FUNCTION_BLOCK WoodBunkEx
VAR_IN_OUT //controls
	execute : BOOL;
	stop : BOOL;
	
	manualStep : BOOL;
	manualSuction : BOOL;
END_VAR
VAR_IN_OUT //references to required hardware
	robotLeft, robotRight : RobotA21;
	toolStorageLeft, toolStorageRight : A21ToolStorage;
	
	stagingTableLeft, stagingTableRight : StagingTable;
	magazineLeft, magazineRight : SkidMagazine;
	
	strapper : StrapMachine;
	
	horizontalDriveLeft, horizontalDriveRight : AirPiston;
	verticalDriveLeft, verticalDriveRight : ClearLinkMC;
	pistonBottom : SimplePiston;
	
	suctionTop : ARRAY[*] OF SuctionPad; (*1..3*)
	suctionLeft : ARRAY[*] OF SuctionPad; (*1..4*)
	suctionRight : ARRAY[*] OF SuctionPad; (*1..4*)
	suctionBottom : ARRAY[*] OF SuctionPad; (*1..2*)
END_VAR
VAR_OUTPUT
	//ready : BOOL;
	done : BOOL;
	
	generalError : BOOL;
	errorLeft, errorRight : BOOL;
END_VAR
VAR //for testing, to be removed when deployoed
	latchLeft, latchRight : BOOL; //prevents SMC sliders from overshooting the inner limit sensor
	
	suctionEnableTop : BOOL;
	suctionEnableLeft : BOOL;
	suctionEnableRight : BOOL;
	suctionEnableBottom : BOOL;
END_VAR
VAR	
	topSuctionDelay : TON;
	
	step : (IDLE, STAGING, LOAD_WB, PUSH, STRAP, RELEASE, COMPLETE := 1050);
	iPair : INT;
	//these 2 ints should replace the 4 ints after
	masterStep : INT;
	subStepLeft, subStepRight : INT;
	
	loadSet : INT;
	loadStepLeft, loadStepRight : INT;
	
	stageSet : INT;	
	stageStepLeft, stageStepRight : INT;
	iSlotLeft, iSlotRight : INT;
END_VAR
VAR //local types
	demoHeight : REAL := 600; //mm
	materialsArr : ARRAY[0..GVL.maxPairs] OF PositionMaterials := [
		(
			position := 0,
			top := 'WDS20', left := 'WDS20', right := 'WDS20', bottom := 'WDB20'
		),
		(
			position := 69,
			top := 'WDS20', left := 'WDS20', right := 'WDS20', bottom := 'WDB20'
		)];
	
	templateSlotsLeft, templateSlotsRight : ARRAY[1..10] OF STRING;
	templateOccupancyLeft, templateOccupancyRight : ARRAY[1..10] OF BOOL;
	stagingTemplateLeft, stagingTemplateRight AT %M* : StagingTable;	
	stagingArrayLeft, stagingArrayRight : ARRAY[0..(GVL.maxPairs+1)*2] OF STRING;
	
	insertionLeft, insertionRight : Insertion;
	loadedMaterials : ARRAY[Surface.TOP..Surface.BOTTOM] OF STRING;
END_VAR
VAR CONSTANT
	sectionID : SectionEnum := SectionEnum.WOOD_BUNK;
END_VAR
VAR
	a,b,c,d : BOOL;
	suctionTimerLeft, suctionTimerRight : TON;
END_VAR

callLocalModules(); //initialize local modules

IF stop THEN
	stopSequence(); //stop everything
	RETURN;
END_IF
(*
IF NOT insertionLeft.screw.HomeSet OR NOT insertionRight.screw.HomeSet THEN
	homingSequence(); //homing all motion devices and robots
	RETURN;
END_IF
*)
a S= suctionTop[1].occupied AND suctionTop[2].occupied AND suctionTop[3].occupied;
b S= suctionLeft[1].occupied AND suctionLeft[2].occupied AND suctionLeft[3].occupied AND suctionLeft[4].occupied;
c S= suctionRight[1].occupied AND suctionRight[2].occupied AND suctionRight[3].occupied AND suctionRight[4].occupied;
d S= suctionBottom[1].occupied AND suctionBottom[2].occupied;

CASE step OF
	IDLE:
		IF execute THEN
			execute := FALSE;
			suctionEnableTop := suctionEnableLeft := suctionEnableRight := suctionEnableBottom := FALSE;
			step := STAGING;
		END_IF
		
		SetSuctions(suctionTop, suctionEnableTop);
		SetSuctions(suctionLeft, suctionEnableLeft);
		SetSuctions(suctionRight, suctionEnableRight);
		SetSuctions(suctionBottom, suctionEnableBottom);
		
	STAGING:
		IF NOT done THEN
			done := stage(error => generalError);
		END_IF
		
		IF
			(manualStep AND_THEN execute) OR
			(NOT manualStep AND_THEN done)
		THEN
			execute := FALSE;
			done := FALSE;
			step := LOAD_WB;
		END_IF
	
	LOAD_WB:
		IF NOT done THEN
			done := load(pairIndex := iPair, error => generalError);
		END_IF
		
		IF manualSuction THEN
			SetSuctions(suctionTop, suctionEnableTop);
			SetSuctions(suctionLeft, suctionEnableLeft);
			SetSuctions(suctionRight, suctionEnableRight);
			SetSuctions(suctionBottom, suctionEnableBottom);
		END_IF
		
		IF
			(manualStep AND_THEN execute) OR
			(NOT manualStep AND_THEN done)
		THEN
			done := FALSE;
			suctionEnableTop := suctionEnableLeft := suctionEnableRight := suctionEnableBottom := FALSE;
			execute := FALSE;
			
			step := PUSH;
		END_IF
		
	PUSH:
		IF
			(manualStep AND_THEN execute) OR
			(latchLeft AND latchRight AND pistonBottom.extended)
		THEN
			latchLeft := latchRight := FALSE;
			execute := FALSE;
			step := STRAP;
			RETURN;
		END_IF
		
		IF NOT validateSuctionQuality(checkTop:= TRUE, checkLeft:= TRUE, checkRight:= FALSE, checkBottom:= FALSE) THEN
			generalError := TRUE;
			RETURN;
		END_IF
		(*
		IF 
			insertionLeft.sliderPos <> demoHeight/2 //OR 
			//insertionRight.sliderPos <> demoHeight/2 //OR 
			//NOT insertionBottom.contact
		THEN
			insertionLeft.slideAbsolute(demoHeight/2);
			//insertionRight.slideAbsolute(demoHeight/2);
			RETURN;
		END_IF
		*)
		
		IF insertionLeft.screw.AtInnerLimit THEN
			latchLeft := TRUE;
		ELSIF NOT latchLeft THEN
			insertionLeft.press();
		END_IF
		
		IF insertionRight.screw.AtInnerLimit THEN
			latchRight := TRUE;
		ELSIF NOT latchRight THEN
			insertionRight.press();
		END_IF
		pistonBottom.extend();
		
	STRAP:
		topSuctionDelay(IN:= , PT:= T#1S, Q=> , ET=> );
		
		strapper.bEnable := TRUE;
		IF strapper.done THEN
			topSuctionDelay.IN := FALSE;
			step := RELEASE;
			RETURN;
		END_IF
		
		IF topSuctionDelay.Q THEN
			SetSuctions(suctionTop, FALSE);
			SetSuctions(suctionLeft, FALSE);
			SetSuctions(suctionRight, FALSE);
			SetSuctions(suctionBottom, FALSE);
		ELSIF strapper.atBundleLevel THEN
			topSuctionDelay.IN := TRUE;
		END_IF
		
		IF strapper.ready THEN
			strapper.strap();
		END_IF
		
		IF execute THEN
			topSuctionDelay.IN := FALSE;
			execute := FALSE;
			step := RELEASE;
		END_IF
		
	RELEASE: //release command		
		//insertionLeft.slideAbsolute(0);
		//insertionRight.slideAbsolute(0);
		
		insertionLeft.release();
		insertionRight.release();
		pistonBottom.retract();
		
		IF 
			(insertionLeft.screw.AtHome AND insertionRight.screw.AtHome AND pistonBottom.retracted) OR
			execute
		THEN
			execute := FALSE;
			step := COMPLETE;
		END_IF
	
	COMPLETE:
		//reset everything
		iPair := (iPair + 1) MOD GVL.maxPairs;
		step := IDLE;
		a := b := c := d := FALSE;
END_CASE

ACTION callLocalModules:
{warning disable C0371}
stagingTemplateLeft(slots := templateSlotsLeft, occupied := templateOccupancyLeft);
stagingTemplateRight(slots := templateSlotsRight, occupied := templateOccupancyRight);

insertionLeft(
	enable:= TRUE, 
	slider:= verticalDriveLeft, 
	screw:= horizontalDriveLeft, 
	contact=> , 
	softContact=> , 
	busy=> , 
	error=> , 
	home=> , 
	homingComplete=> , 
	sliderPos=> );
	
insertionRight(
	enable:= TRUE, 
	slider:= verticalDriveRight, 
	screw:= horizontalDriveRight,  
	contact=> , 
	softContact=> , 
	busy=> , 
	error=> , 
	home=> , 
	homingComplete=> , 
	sliderPos=> );
END_ACTION

METHOD createStagingArrayLeft : BOOL
VAR
	remainingMaterial : STRING;
	splitMaterial : STRING;
	
	i : INT;
END_VAR
FOR i:=0 TO GVL.maxPairs BY 1 DO
	remainingMaterial := materialsArr[i].top;
	WHILE FIND(remainingMaterial, '_') > 0 DO
		splitCombinedMaterials(remainingMaterial, splitMaterial);
		IF splitMaterial <> '' THEN
			AddToStringArray(arr := stagingArrayLeft, newString := splitMaterial, numElements => , nextIndex => );
		END_IF
	END_WHILE
	
	IF remainingMaterial <> '' THEN
		AddToStringArray(arr := stagingArrayLeft, newString := remainingMaterial, numElements => , nextIndex => );
	END_IF
	
	
	remainingMaterial := materialsArr[i].left;
	WHILE FIND(remainingMaterial, '_') > 0 DO
		splitCombinedMaterials(remainingMaterial, splitMaterial);
		IF splitMaterial <> '' THEN
			AddToStringArray(arr := stagingArrayLeft, newString := splitMaterial, numElements => , nextIndex => );
		END_IF
	END_WHILE
	
	IF remainingMaterial <> '' THEN
		AddToStringArray(arr := stagingArrayLeft, newString := remainingMaterial, numElements => , nextIndex => );
	END_IF
END_FOR
END_METHOD

METHOD createStagingArrayRight : BOOL
VAR
	remainingMaterial : STRING;
	splitMaterial : STRING;
	
	i : INT;
END_VAR
FOR i:=0 TO GVL.maxPairs*2 BY 1 DO
	remainingMaterial := materialsArr[i].bottom;
	WHILE FIND(remainingMaterial, '_') > 0 DO
		splitCombinedMaterials(remainingMaterial, splitMaterial);
		IF splitMaterial <> '' THEN
			AddToStringArray(arr := stagingArrayRight, newString := splitMaterial, numElements => , nextIndex => );
		END_IF
	END_WHILE
	
	IF remainingMaterial <> '' THEN
		AddToStringArray(arr := stagingArrayRight, newString := remainingMaterial, numElements => , nextIndex => );
	END_IF
	
	
	
	remainingMaterial := materialsArr[i].right;
	WHILE FIND(remainingMaterial, '_') > 0 DO
		splitCombinedMaterials(remainingMaterial, splitMaterial);
		IF splitMaterial <> '' THEN
			AddToStringArray(arr := stagingArrayRight, newString := splitMaterial, numElements => , nextIndex => );
		END_IF
	END_WHILE
	
	IF remainingMaterial <> '' THEN
		AddToStringArray(arr := stagingArrayRight, newString := remainingMaterial, numElements => , nextIndex => );
	END_IF
END_FOR
END_METHOD

METHOD PROTECTED generateStagingTemplate : BOOL
VAR
	remainingMaterial : STRING;
	splitMaterial : STRING;
	
	i : INT;
END_VAR
VAR_STAT
	temp : INT;
END_VAR
createStagingArrayLeft();
createStagingArrayRight();

//AddToStringArray(arr := stagingArrayLeft, newString := 'WDB20', numElements =>, nextIndex => );

(*
iterate through all pairs and autofill the template
replace succesfully autofilled materials with empty string

when staging needs to be performed a 2nd time, autofilling empty strings is always unsuccessful
*)
FOR i:=0 TO GVL.maxPairs*2 BY 1 DO
	IF stagingTemplateLeft.autofill(materialID := stagingArrayLeft[i]) THEN
		stagingArrayLeft[i] := '';
	END_IF
	
	IF stagingTemplateRight.autofill(materialID := stagingArrayRight[i]) THEN
		stagingArrayRight[i] := '';
	END_IF
END_FOR

(*
stagingTemplateLeft.autofill(demoPairWB.top);
stagingTemplateLeft.autofill(demoPairWB.left);

stagingTemplateRight.autofill(demoPairWB.right);
stagingTemplateRight.autofill(demoPairWB.bottom);
*)

generateStagingTemplate := TRUE;
END_METHOD

ACTION homingSequence:
insertionLeft.homingSequence();
insertionRight.homingSequence();
pistonBottom.retract();
END_ACTION

METHOD PROTECTED load : BOOL
VAR_INPUT
	pairIndex : INT;
END_VAR
VAR_OUTPUT
	error : BOOL;
END_VAR
VAR
	pair : REFERENCE TO PositionMaterials REF= materialsArr[pairIndex];
END_VAR
{warning disable C0371}

IF robotLeft.error OR robotRight.error THEN
	error := TRUE;
	RETURN;
	
ELSIF NOT robotLeft.reserve(sectionID) OR NOT robotRight.reserve(sectionID) THEN //loading requires both robots be reserved together
	RETURN;
	
ELSIF //robots have wrong tool
	(robotLeft.tool <> sectionID AND_THEN NOT robotLeft.changeEOAT(targetTool := sectionID)) OR
	(robotRight.tool <> sectionID AND_THEN NOT robotRight.changeEOAT(targetTool := sectionID))
THEN
	RETURN;
END_IF

CASE loadSet OF
	0: //top and bottom
		IF 
			loadingSequence(
				robot:= robotLeft, 
				table:= stagingTableLeft, 
				loadStep:= loadStepLeft, 
				slot:= iSlotLeft,
				suctions:= suctionTop,
				suctionTimer:= suctionTimerLeft,
				surfaceID:= Surface.TOP, 
				material:= pair.top, 
				fail=> errorLeft)
			
			AND
			loadingSequence(
				robot:= robotRight,
				table:= stagingTableRight, 
				loadStep:= loadStepRight, 
				slot:= iSlotRight,
				suctions:= suctionBottom,
				suctionTimer:= suctionTimerRight,
				surfaceID:= Surface.BOTTOM, 
				material:= pair.bottom, 
				fail=> errorRight)
			
		THEN
			suctionTimerLeft.IN := suctionTimerRight.IN := FALSE;
			loadStepLeft := loadStepRight := 0;
			loadSet := 10;
		END_IF
		
	10: //sides
		IF
			loadingSequence(
				robot:= robotLeft, 
				table:= stagingTableLeft, 
				loadStep:= loadStepLeft, 
				slot:= iSlotLeft,
				suctions:= suctionLeft,
				suctionTimer:= suctionTimerLeft,
				surfaceID:= Surface.LEFT, 
				material:= pair.left, 
				fail=> errorLeft)
			
			AND
			loadingSequence(
				robot:= robotRight, 
				table:= stagingTableRight, 
				loadStep:= loadStepRight, 
				slot:= iSlotRight,
				suctions:= suctionRight,
				suctionTimer:= suctionTimerRight,
				surfaceID:= Surface.RIGHT, 
				material:= pair.right, 
				fail=> errorRight)
		THEN
			suctionTimerLeft.IN := suctionTimerRight.IN := FALSE;
			loadStepLeft := loadStepRight := 0;
			loadSet := COMPLETE;
		END_IF
		
	COMPLETE:
		suctionTimerLeft.IN := suctionTimerRight.IN := FALSE;
		
		loadSet := 0;
		loadStepLeft := loadStepRight := 0;
		
		robotLeft.release(sectionID);
		robotRight.release(sectionID);
		
		load := TRUE;
END_CASE
END_METHOD

METHOD loadingSequence : BOOL
VAR_IN_OUT
	robot : RobotA21;
	table : StagingTable;
	suctions : ARRAY[*] OF SuctionPad;
	loadStep : INT;
	slot : INT;
	
	suctionTimer : TON;
END_VAR
VAR_INPUT
	surfaceID : Surface;
	material : STRING;
END_VAR
VAR_OUTPUT
	fail : BOOL;
END_VAR
VAR
	recoveryMagazine : REFERENCE TO SkidMagazine;
	recoveryStageStep : REFERENCE TO INT;
	suctionDelay : TIME := T#2S;
END_VAR
{warning disable C0371}
IF material = '' THEN
	robot.clearCommand();
	loadingSequence := TRUE;
	RETURN;
END_IF

CASE loadStep OF
	0: //wait for robot
		robot.clearCommand();
		IF robot.Ready THEN
			loadStep := 10;
			slot := 0;
		END_IF
		
	10: //grab from table
		IF slot < 1 AND_THEN NOT table.findSlot(materialID := material, atPosition => slot) THEN 
			fail := TRUE;
			RETURN;
		END_IF
		
		IF NOT table.isOccupied(i := slot) AND table.getSlot(i := slot) <> '' THEN //move from table to robot gripper
			robot.HoldMaterial := table.getSlot(i := slot);
			table.remove(i := slot, materialID => );
		END_IF
		
		IF robot.Done THEN
			loadStep := COMPLETE;
			RETURN;
		ELSIF robot.materialAtHoldingPosition >= 1 AND robot.materialAtHoldingPosition <= 8 THEN
			loadStep := 20;
			RETURN;
		END_IF
		
		CASE surfaceID OF
			Surface.TOP: 					robot.setGroup(group := 1, value := A21.LOAD_BUNK_TOP); 
			Surface.LEFT, Surface.RIGHT: 	robot.setGroup(group := 1, value := A21.LOAD_BUNK_SIDE);
			Surface.BOTTOM: 				robot.setGroup(group := 1, value := A21.LOAD_BUNK_BOTTOM);
		END_CASE
		robot.setGroup(group := 2, value := slot); 
			
	20: //place to insertion
		IF robot.materialAtHoldingPosition > 0 AND robot.HoldMaterial <> '' THEN //move from gripper to insertion
			IF loadedMaterials[surfaceID] = '' THEN //transfer to insertion as is
				loadedMaterials[surfaceID] := robot.HoldMaterial;
			ELSE //join with existing material using underscore _
				loadedMaterials[surfaceID] := JoinStrings(loadedMaterials[surfaceID], robot.HoldMaterial, '_');
			END_IF
			robot.HoldMaterial := '';
		END_IF
		
		CASE surfaceID OF
			Surface.TOP, Surface.BOTTOM:
				SetSuctions(suctions, TRUE (*robot.materialAtHoldingPosition = 1 OR robot.materialAtHoldingPosition = 4*));
				
			Surface.LEFT, Surface.RIGHT:
				SetSuctions(suctions, TRUE (*robot.materialAtHoldingPosition = 2 OR robot.materialAtHoldingPosition = 3*));
				(*
				FOR i:=LOWER_BOUND(suctions, 1) TO UPPER_BOUND(suctions, 1) BY 1 DO
					
					IF i < UPPER_BOUND(suctions, 1)/2 THEN
						suctions[i].enable := robot.materialAtHoldingPosition = 2; //enable upper half suctions
					ELSE
						suctions[i].enable := robot.materialAtHoldingPosition = 3; //enable lower half suctions
					END_IF

				END_FOR
				*)
		END_CASE
		
		suctionTimer(IN:= , PT:= suctionDelay, Q=> , ET=> );
		suctionTimer.IN := TRUE;
		IF NOT suctionTimer.Q THEN
			RETURN;
		END_IF
		
		IF robot.Done THEN
			suctionTimer.IN := FALSE;
			loadStep := COMPLETE;
		END_IF
		
		robot.setGroup(group := 9, value := robot.materialAtHoldingPosition);
	
	COMPLETE:
		robot.clearCommand();
		
		//check insertion quality
		suctionTimer(IN:= , PT:= suctionDelay, Q=> , ET=> );
		suctionTimer.IN := TRUE;
		IF NOT suctionTimer.Q THEN
			RETURN;
		END_IF
		
		IF InsertionQuality(suctions := suctions, insertionMaterial := loadedMaterials[surfaceID], recipeMaterial := material) THEN
			loadingSequence := TRUE;
		ELSE //recovery - remove, restage, and reload
			suctionTimer.IN := FALSE;
			loadStep := 100;
			
		END_IF
		
	100:
		robot.clearCommand();
		IF robot.Ready THEN
			loadStep := 110;
		END_IF
		
	110: //recovery - remove from insertion
		IF robot.Done THEN
			loadStep := 120;
			RETURN;
		END_IF
		
		CASE surfaceID OF
			Surface.TOP:					robot.setGroup(group := 1, value := A21.REMOVE_BUNK_TOP);
			Surface.LEFT, Surface.RIGHT:	robot.setGroup(group := 1, value := A21.REMOVE_BUNK_SIDE);
			Surface.BOTTOM:					robot.setGroup(group := 1, value := A21.REMOVE_BUNK_BOTTOM);
		END_CASE
		
	120:
		robot.clearCommand();
		IF robot.Ready THEN
			loadStep := 130;
		END_IF
		
	130: //recovery - restage
		CASE surfaceID OF
			Surface.TOP, Surface.LEFT:
				recoveryMagazine REF= magazineLeft;			
				recoveryStageStep REF= stageStepLeft;
				
			Surface.RIGHT, Surface.BOTTOM:
				recoveryMagazine REF= magazineRight;			
				recoveryStageStep REF= stageStepRight;
				
		END_CASE
		
		IF
			stageSingle(
				robot:= robot, 
				table:= table, 
				magazine:= recoveryMagazine, 
				stageStep:= recoveryStageStep, 
				slot:= slot, 
				material:= material, 
				fail=> fail)
		THEN
			SetSuctions(suctionPads := suctions, state := FALSE);
			loadStep := 0; //retry
		END_IF
	
END_CASE
END_METHOD

METHOD splitCombinedMaterials : BOOL
VAR_IN_OUT
	materialID : STRING;
	splitMaterial : STRING;
END_VAR
VAR
	i : INT;
END_VAR
FindAndSplitChar(
	sSeparatorChar:= '_', 
	pSrcString:= ADR(materialID), 
	
	pLeftString:= ADR(splitMaterial), 
	nLeftSize:= SIZEOF(splitMaterial), 
	
	pRightString:= ADR(materialID), 
	nRightSize:= SIZEOF(materialID), 
	
	bSearchFromRight:= FALSE);
END_METHOD

METHOD stage : BOOL
VAR_OUTPUT
	error : BOOL;
END_VAR
VAR_STAT
	temp : ARRAY[1..4] OF BOOL;
	boundsErr : ARRAY[1..4] OF BOOL;
END_VAR
{warning disable C0371}
temp[1] := stagingTableLeft.isOccupied(i := 1, errorBounds => boundsErr[1]);
temp[2] := stagingTableLeft.isOccupied(i := 2, errorBounds => boundsErr[2]);
temp[3] := stagingTableLeft.isOccupied(i := 3, errorBounds => boundsErr[4]);
temp[4] := stagingTableLeft.isOccupied(i := 4, errorBounds => boundsErr[3]);

CASE stageSet OF
	0: //create staging template
		IF generateStagingTemplate() THEN
			stageSet := 10;
		END_IF
	
	10: //staging sequence
		IF
			stagingSequence(				
				robot:= robotLeft, 
				template:= stagingTemplateLeft,
				table:= stagingTableLeft,  
				magazine:= magazineLeft, 
				stageStep:= stageStepLeft, 
				iSlot:= iSlotLeft,
				error=> errorLeft)
			
			AND
			stagingSequence(
				robot:= robotRight, 
				template:= stagingTemplateRight, 
				table:= stagingTableRight, 
				magazine:= magazineRight, 
				stageStep:= stageStepRight, 
				iSlot:= iSlotRight,
				error=> errorRight)
		THEN
			stageStepLeft := stageStepRight := 0;
			iSlotLeft := iSlotRight := 0;
			
			stageSet := COMPLETE;
		END_IF
		
	COMPLETE:
		stagingTemplateRight.clear(); //clear the staging templates
		stagingTemplateLeft.clear();
		
		robotLeft.release(sectionID); //release the robots
		robotRight.release(sectionID);
		
		stageSet := 0;
		stage := TRUE;
		
END_CASE
END_METHOD

METHOD stageSingle : BOOL
VAR_IN_OUT
	robot : RobotA21;
	table : StagingTable;
	magazine : SkidMagazine;
	stageStep : INT;
END_VAR
VAR_INPUT
	slot : INT;
	material : STRING;
END_VAR
VAR_OUTPUT
	fail : BOOL;
END_VAR
VAR
	column : INT; //valid positions start from 1
END_VAR
VAR CONSTANT
	suctionDistance : INT := 10;
END_VAR
{warning disable C0371}
{warning disable C0195}
(*
this method allows the staging of single bunks without the use of a template
neccessary for restaging bunks that are not loaded properly into insertions
*)

IF
	material = '' OR_ELSE
	table.getSlot(i := slot) = material
THEN
	robot.clearCommand();
	stageSingle := TRUE;
	RETURN;
END_IF

//follow the template as is
CASE stageStep OF
	0:
		robot.clearCommand();
		IF robot.Ready THEN
			stageStep := 10;
		END_IF
		
	10: //grab from magazine
		IF NOT magazine.findSlot(materialID := material, atPosition => column) THEN
			fail := TRUE;
			RETURN;
		END_IF
		
		IF robot.eoatDistance < suctionDistance THEN //robot is grabbing material
			robot.HoldMaterial := magazine.getSlot(i := column);
		END_IF
		
		IF robot.Done THEN
			stageStep := COMPLETE;
			RETURN;
		ELSIF table.isOccupied(slot) THEN //wood bunk registered on table
			stageStep := 20;
			RETURN;
		END_IF
		
		robot.setGroup(group := 1, value := A21.STAGE_BUNK);
		robot.setGroup(group := 2, value := column);
		robot.setGroup(group := 3, value := slot);
	
	20: //place to table
		IF
			table.isOccupied(slot) AND //staging table slot is occupied
			table.getSlot(slot) = '' AND //staging table has not recorded a bunk
			robot.HoldMaterial <> '' //robot is carrying a bunk
		THEN //move material from robot to table
			table.place(i := slot, materialID := robot.HoldMaterial);
			robot.HoldMaterial := '';
		END_IF
		
		IF robot.Done THEN
			stageStep := COMPLETE;
			RETURN;
		END_IF
	
	COMPLETE: //check here if staging is successful or needs to be repeated
		//if the material is registered on the table, this step will not be evaluated due to the guard clause above
		robot.clearCommand();
		
		IF table.isOccupied(slot) AND table.getSlot(i := slot) = material THEN
			stageSingle := TRUE;
		ELSE
			table.remove(i := slot, materialID => );
			stageStep := 0;
		END_IF
		
END_CASE
END_METHOD

METHOD stageSingleV2 : BOOL
VAR_IN_OUT
	robot : RobotA21;
	table : StagingTable;
	magazine : SkidMagazine;
	stageStep : INT;
END_VAR
VAR_INPUT
	slot : INT;
	material : STRING;
END_VAR
VAR_OUTPUT
	error : BOOL;
END_VAR
VAR
	column : INT; //valid positions start from 1
END_VAR
VAR CONSTANT
	suctionDistance : INT := 10;
END_VAR
{warning disable C0371}
{warning disable C0195}
(*
this method allows the staging of single bunks without the use of a template
neccessary for restaging bunks that are not loaded properly into insertions
*)

IF material = '' THEN
	robot.clearCommand();
	stageSingleV2 := TRUE;
	RETURN;
END_IF

//follow the template as is
CASE stageStep OF
	0:
		robot.clearCommand();
		IF robot.Ready THEN
			stageStep := 10;
		END_IF
		
	10: //move from magazine to table
		IF NOT magazine.findSlot(materialID := material, atPosition => column) THEN
			error := TRUE;
			RETURN;
		END_IF
		
		IF robot.eoatDistance < suctionDistance THEN //robot is grabbing material
			robot.HoldMaterial := magazine.getSlot(i := column);
		END_IF
		
		IF robot.Done THEN
			stageStep := COMPLETE;
			RETURN;
		END_IF
		
		robot.setGroup(group := 1, value := A21.STAGE_BUNK);
		robot.setGroup(group := 2, value := column);
		robot.setGroup(group := 3, value := slot);

	COMPLETE: //check here if staging is successful or needs to be repeated
		robot.clearCommand();
		
		IF table.isOccupied(i := slot) THEN
			table.place(i := slot, materialID := robot.HoldMaterial);
			stageSingleV2 := TRUE;
		ELSE
			stageStep := 0;
			error := TRUE;
		END_IF
		
		robot.HoldMaterial := '';
END_CASE
END_METHOD

METHOD stagingSequence : BOOL
VAR_IN_OUT
	robot : RobotA21;
	template : StagingTable;
	table : StagingTable;
	magazine : SkidMagazine;
	stageStep : INT;
	iSlot : INT;
END_VAR
VAR_OUTPUT
	error : BOOL;
END_VAR
VAR
	magazineColumn : INT; //valid positions start from 1
END_VAR
VAR CONSTANT
	(*
	WIP : INT := 0;
	PASSED : INT := 1;
	FAILED : INT := 2;
	*)
	suctionDistance : INT := 10;
END_VAR
VAR_STAT
	tempMaterial : STRING;
	tempOccupied : BOOL;
	temp : BOOL;
	
	adr1, adr2 : PVOID;
END_VAR
{warning disable C0371}
{warning disable C0195}

IF iSlot = 0 THEN
	iSlot := 1;
	RETURN;
ELSIF table.isFull() OR iSlot > 10 THEN //staging table is full or all slots have been iterated through
	robot.clearCommand();
	robot.release(sectionID);
	stagingSequence := TRUE;
	RETURN;
END_IF

IF robot.error THEN
	error := TRUE;
	RETURN;
ELSIF robot.reservation <> sectionID AND_THEN NOT robot.reserve(sectionID) THEN
	RETURN;
ELSIF robot.tool <> sectionID AND_THEN NOT robot.changeEOAT(targetTool := sectionID) THEN
	RETURN;
END_IF

//follow the template as is
IF
	stageSingleV2(
		robot:= robot, 
		table:= table, 
		magazine:= magazine, 
		stageStep:= stageStep, 
		slot:= iSlot, 
		material:= template.getSlot(iSlot), 
		error=> error)
THEN
	iSlot := iSlot + 1;
	stageStep := 0;
END_IF
END_METHOD

ACTION stopSequence:
insertionLeft.stop();
insertionRight.stop();
pistonBottom.stop();

robotLeft.clearCommand();
robotRight.clearCommand();

//stop conveyors
END_ACTION

METHOD validateSuctionQuality : BOOL
VAR_INPUT
	checkTop : BOOL;
	checkLeft : BOOL;
	checkRight : BOOL;
	checkBottom : BOOL;
END_VAR
validateSuctionQuality := 
	(
		NOT checkTop OR_ELSE InsertionQuality(
			suctions:= suctionTop, 
			insertionMaterial:= loadedMaterials[Surface.TOP], 
			recipeMaterial:= materialsArr[iPair].top)
	) AND
	(
		NOT checkLeft OR_ELSE InsertionQuality(
			suctions:= suctionLeft, 
			insertionMaterial:= loadedMaterials[Surface.LEFT], 
			recipeMaterial:= materialsArr[iPair].left)
	) AND
	(
		NOT checkRight OR_ELSE InsertionQuality(
			suctions:= suctionRight, 
			insertionMaterial:= loadedMaterials[Surface.RIGHT], 
			recipeMaterial:= materialsArr[iPair].right)
	) AND
	(
		NOT checkBottom OR_ELSE InsertionQuality(
			suctions:= suctionBottom, 
			insertionMaterial:= loadedMaterials[Surface.BOTTOM], 
			recipeMaterial:= materialsArr[iPair].bottom)
	);
END_METHOD

END_FUNCTION_BLOCK

(* stored: Version 1.1.0.1, ProductVersion 3.1.4024.11
   POU WoodBunkEx: Id {7c192e4b-e9ee-4c1c-a070-15e2c6191789}, SpecialFunc None
   Folder Loading: Id {d5b5a4e4-ee29-48b3-b5c8-451836b38fcb}
   Folder Staging: Id {d65a2989-4fa8-4947-a8e8-602f97dc611d}
   Folder Template: Id {cd893e68-3f3a-4606-a79f-9e9ae0341cae}
   Action callLocalModules: Id {8b2708ac-6691-4038-ae66-c4869c7fa2e2}
   Method createStagingArrayLeft: Id {267fdecb-2bd1-4d34-885b-8346cf63d26a}
   Method createStagingArrayRight: Id {16356a3e-786d-4de1-9a22-49e2a7eb3ddd}
   Method generateStagingTemplate: Id {559e2100-9d18-4e6d-a37b-fe2e4a5b8bd4}
   Action homingSequence: Id {7653a770-9078-4c2c-aad4-1564dbc9f3b2}
   Method load: Id {41d6aef3-60c1-439a-bdd2-e372cfed0011}
   Method loadingSequence: Id {b6930bdc-6b37-4ccd-8367-4e887d0b238c}
   Method splitCombinedMaterials: Id {253040a1-6112-4088-b271-b912c88ba0a3}
   Method stage: Id {394ea3b0-a477-4afc-b551-89e83b2984a7}
   Method stageSingle: Id {f5e1059d-c963-4087-8934-2509cfe03bd5}
   Method stageSingleV2: Id {2d96c33a-964e-4ebf-9f5e-ea6263dc3c9e}
   Method stagingSequence: Id {1cf9906f-6300-40ae-8532-5d125199aeba}
   Action stopSequence: Id {aa2cff5b-4063-4180-a68f-c8e049a6e342}
   Method validateSuctionQuality: Id {b1904323-60a7-4bcf-ac74-c2042e21b0b7} *)
